FUNCTION_BLOCK FB_ComponentChild EXTENDS FB_Component
VAR_INPUT
END_VAR
VAR_OUTPUT
END_VAR
VAR
	fbComponent:		FB_ComponentEX;
END_VAR

SUPER^();

METHOD PUBLIC M_Call
VAR_INPUT
END_VAR
SUPER^.M_Call();

fbComponent.M_Call();
END_METHOD

METHOD PROTECTED M_Initialise : BOOL;
VAR_INPUT
END_VAR
fbObserver.M_Attach(fbComponent);
fbComponent.P_Observer.M_Attach(THIS^);

M_Initialise:= super^.M_Initialise();
END_METHOD

METHOD PROTECTED M_Starting : BOOL
VAR_INPUT
END_VAR
M_Starting:= super^.M_Starting() and fbComponent.M_Request(E_Request.Start);
END_METHOD

END_FUNCTION_BLOCK

(* stored: Version 1.1.0.1, ProductVersion 3.1.4024.12
   POU FB_ComponentChild: Id {ad9f1548-4ce5-024e-1f0d-72220a1fdbb1}, SpecialFunc None
   Method M_Call: Id {3011bb02-ac52-0e83-1df7-8050a651d1e3}
   Method M_Initialise: Id {f6ab3841-4279-0477-217f-e5cb4c5c69c2}
   Method M_Starting: Id {38ddd15f-7483-0cfa-19c2-0690c6226f70} *)
